FUNCTION_BLOCK CL_AxisL2RightBack EXTENDS CL_AxisRobot
var
END_VAR

SUPER^();

METHOD PROTECTED InitDefect : BOOL
sWhichAxis := 'right(L2)-back';
InitDefect := true;
END_METHOD

METHOD PROTECTED InitParams : BOOL
VAR_INPUT
END_VAR
InitParams := super^.InitParams();
_lrInverse := -1.0;
END_METHOD

END_FUNCTION_BLOCK

(* stored: Version 1.1.0.1, ProductVersion 3.1.4024.12
   POU CL_AxisL2RightBack: Id {9581f397-500f-4bc2-83c1-3fff25c338cc}, SpecialFunc None
   Method InitDefect: Id {255aed50-cbe1-4d37-a724-ff92b8ae219e}
   Method InitParams: Id {f630f93c-65da-4341-ab5f-5ba2af850e86} *)
